(* CODESYS project PLC_Training_Estrusora_V3.project

Project tree, tasks and I/O mapping:
  Device : CODESYS Control Win V3 x64, CODESYS, version 3.5.21.40
    application Application
      libraries: Standard, 3.5.18.0 (System); VisuDialogs, * (System)
      task VISU_TASK (cyclic, interval 100 ms, priority 31) calls VisuElems.Visu_Prg
      task MainTask (cyclic, interval t#20ms, priority 1) calls PLC_Main
      function block FB_Inputs [LD]
      visualisation Visualization
      function block FB_Outputs [LD]
      function block FB_Process [LD]
      function block FB_Control [ST]
      function block FB_Events [ST]
      function block FB_PlantSim [ST]
      program PLC_Main [LD]
      global variables GVL_IO
      function block FB_Interlocks [LD]
      function block FB_Recipes [ST]
      text list TextList
      function block FB_LotHistory [ST]
      data type ST_LotRecord
  text list GlobalTextList
  text list System
  function block FB_Interlocks [LD]
*)

// Device/Application/ST_LotRecord
TYPE ST_LotRecord :
STRUCT
	LotNumber : DINT;
    RecipeID : INT;
    RecipeName : STRING[20];
    ProcessTime : TIME;
    MotorSpeed : INT;
    Completed : BOOL;
	CompletionDT : DT;
	TimestampText: STRING := DT_TO_STRING(CompletionDT);
END_STRUCT
END_TYPE

// Device/Application/GVL_IO
VAR_GLOBAL
	
    // =========================
    // RAW INPUTS (simulados / HMI)
    // =========================
	
    StartPB     : BOOL;   // Botón Start (RAW)
    StopPB_NC   : BOOL := TRUE;   // Botón Stop NC (RAW) -> TRUE = circuito OK, FALSE = presionado/abierto
	ResetPB     : BOOL;   // Boton de reset de falla
	LoadHopperPB : BOOL;  //Carga de la tolva
	AutoSelect : BOOL := TRUE;  // Boton del seleccion HMI
	ManualRunPB   : BOOL;  //Boton Arranque manual
	
    Sensor1     : BOOL;   // Sensor de Carga Minima (RAW)
	Sensor2		: BOOL;   //Sensor de carga media (RAW)
	Sensor3     : BOOL;   //Sensor de Carga Maxima (RAW)
	MotorFB     : BOOL;   // Feedback de motor/contactor (simulado)
	
	// =========================
    // NORMALIZED INPUTS (para lógica)
    // =========================
	
    Start       : BOOL;   // Evento/estado usable por lógica
    StopOK      : BOOL;   // TRUE = permitido (stop sano)
	ResetCmd       : BOOL;   // Reset de falla (simulado)
	ManualRunCmd  : BOOL; // Comando de arranque del motor
	LoadHopperCmd : BOOL; // Comando de carga de la tolva
	
	LevelLow    : BOOL;   // Sensor de carga de la tolva minima
	LevelMid    : BOOL;   // Sensor de carga de la tolva Media
	LevelHigh   : BOOL;   // Sensor de carga de la tolva Maximo
	
	// =========================
    // EVENTS (pulsos 1-scan)
    // =========================
	
    Start_Rise   : BOOL;   // Pulso flanco subida Start
    Stop_Fall   : BOOL;   // Pulso flanco bajada StopOK (o StopPB_NC si lo preferís)
	Reset_Rise  : BOOL;   // Pulso Subido para reset de falla.
	LoadHopper_Rise : BOOL; // Pulso Subida de carga de la tolva

	// =========================
    // MODOS / CONTROL
    // =========================
	
	AutoMode : BOOL := TRUE;
	ManualMode : BOOL := FALSE;

	RunCmd       : BOOL;     // Comando general de marcha
	State : INT := 0;        // 0= IDLE, 5=Manual, 10=STARTING, 20=Processing, 40=Complete 90=FAULT
	StateText : STRING[50];	 // almacena la cadena segun estado
	StateProcessing : BOOL;  //Badera de control de estado
	BatchComplete : BOOL;    //Indicador del final del proceso
	
	//==========================
	//Codigos de falla Y alarmas
	//=========================
	
	Fault        : BOOL;  // Falla activa (latch)
	FaultCode_MotorNoStart : BOOL; 
	FaultCode_LevelInvalid : BOOL; 
	
	Alarm_NoMaterial_Latched : BOOL; // Latch de control de Alarmas
	Alarm_NoMaterialStart : BOOL;
	AlarmText : STRING[50];
	
    // =========================
    // OUTPUTS (lógicos)
    // =========================
	
	AlarmLamp    : BOOL;  // Lámpara/alarma (lógico Rojo)
    MotorCmd     : BOOL;  // Comando a motor (lógico)
    ReadyLamp    : BOOL;   // Lampara de Maquina Lista para correr (Logico Amarillo)
	
	//==========================
	// Simulacion / Proceso
	//==========================
	
	SimEnable  : BOOL := TRUE;   // habilita simulación de planta
    MotorAngle : INT  := 0;      // 0..359 (para animación)
	ProcessTimeA : TIME ;  //Tiempo del proceso por receta.
	CantLotesProc   : DINT;      //Cuenta la cantidad de lotes procesados
	VelocidadMotor : INT; //Velocidad de giro del motor
	
	//==========================
	//Interlocks
	//==========================
	
	StartPermissive : BOOL ;
	RunPermissive : BOOL ;
	LoadPermissive : BOOL;
	ResetPermissive : BOOL;
	Ready       : BOOL;   // Comando de inicio.
	RecipeChangePermissive: BOOL ; // Limita el cambio de receta durante una corrida.
	
	//==========================
	//Recetas (Variables)
	//==========================

	RecipeSelected : INT; //Recibe la opcion seleccionada
	RecipeID : INT ; //Identificador de la receta.
	RecipeName : STRING[20]; // Recibe el nombre de la receta
	
	//==========================
	//Historial de lotes y fallas
	//==========================
	
	LotHistory : ARRAY[1..20] OF ST_lotRecord;
	LotHistoryIndex : INT := 1;	
	TimestampText : STRING[30];
	LastLotTimestampText : STRING[30];
	LotHistoryCount : INT ;
	
END_VAR

// Device/Application/PLC_Main
PROGRAM PLC_Main
VAR
	fbInputs: FB_Inputs;
	fbEvents: FB_Events;
	fbControl: FB_Control;
	fbProcess: FB_Process;
	fbOutputs: FB_Outputs;
	fbPlantSim: FB_PlantSim;
	fbInterlocks: FB_Interlocks;
	fbRecipes: FB_Recipes;
	fbLotHistory: FB_LotHistory;
	
	VarTimeCur : DT;
	
	Reloj: RTC;
END_VAR

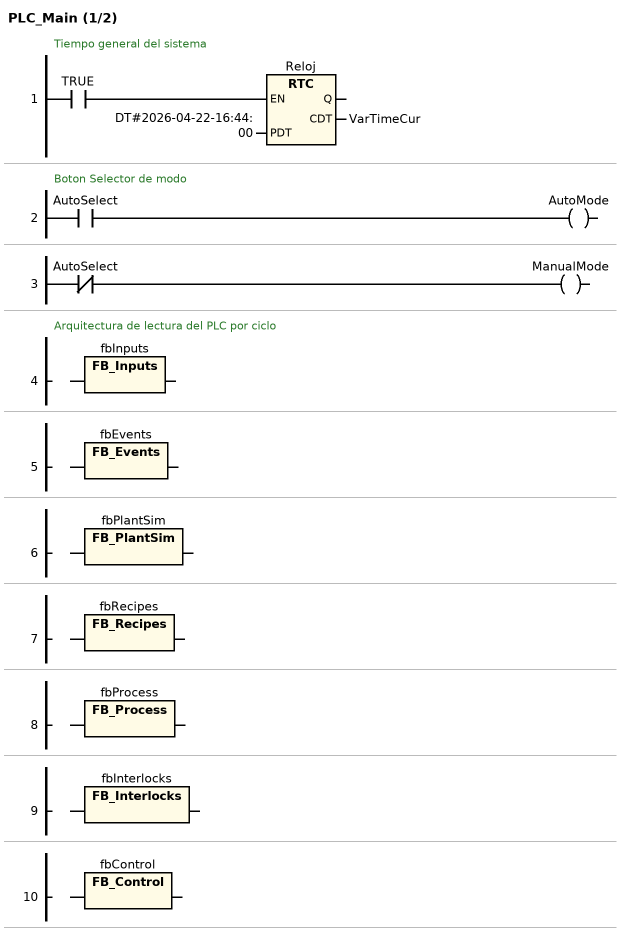
// NETWORK 1
// Tiempo general del sistema
Reloj(EN := TRUE, PDT := DT#2026-04-22-16:44:00, CDT => VarTimeCur); // RTC

// NETWORK 2
// Boton Selector de modo
AutoMode := AutoSelect;

// NETWORK 3
ManualMode := NOT AutoSelect;

// NETWORK 4
// Arquitectura de lectura del PLC por ciclo
fbInputs(); // FB_Inputs

// NETWORK 5
fbEvents(); // FB_Events

// NETWORK 6
fbPlantSim(); // FB_PlantSim

// NETWORK 7
fbRecipes(); // FB_Recipes

// NETWORK 8
fbProcess(); // FB_Process

// NETWORK 9
fbInterlocks(); // FB_Interlocks

// NETWORK 10
fbControl(); // FB_Control

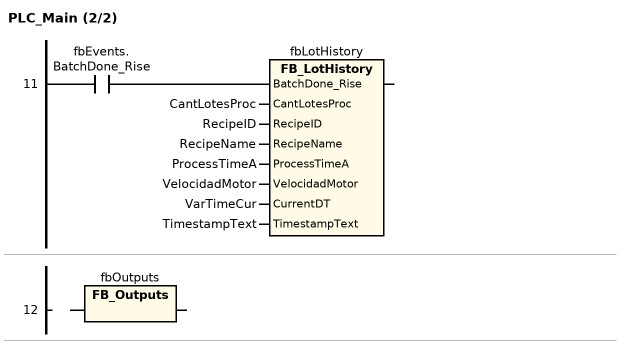
// NETWORK 11
fbLotHistory(
    BatchDone_Rise := fbEvents.BatchDone_Rise,
    CantLotesProc := CantLotesProc,
    RecipeID := RecipeID,
    RecipeName := RecipeName,
    ProcessTimeA := ProcessTimeA,
    VelocidadMotor := VelocidadMotor,
    CurrentDT := VarTimeCur,
    TimestampText := TimestampText); // FB_LotHistory

// NETWORK 12
fbOutputs(); // FB_Outputs

END_PROGRAM

// Device/Application/FB_Inputs
FUNCTION_BLOCK FB_Inputs
VAR_INPUT
END_VAR
VAR_OUTPUT
END_VAR
VAR
END_VAR

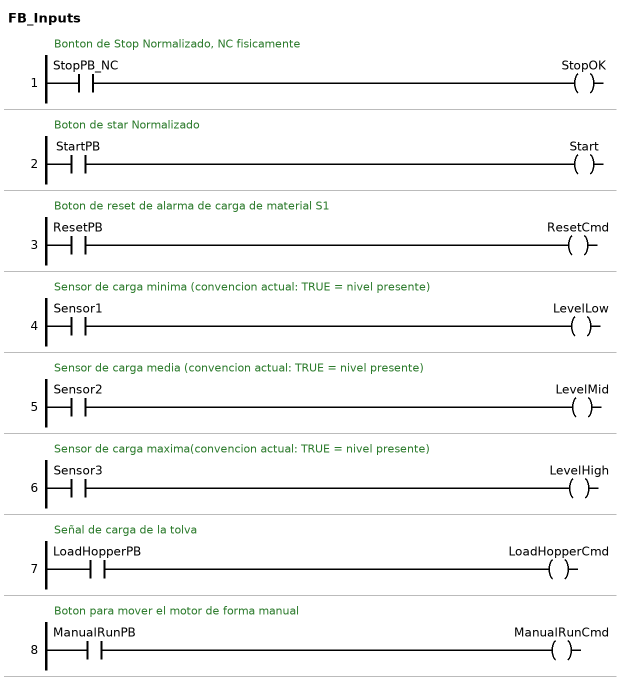
// NETWORK 1
// Bonton de Stop Normalizado, NC fisicamente
StopOK := StopPB_NC;

// NETWORK 2
// Boton de star Normalizado
Start := StartPB;

// NETWORK 3
// Boton de reset de alarma de carga de material S1
ResetCmd := ResetPB;

// NETWORK 4
// Sensor de carga minima (convencion actual: TRUE = nivel presente)
LevelLow := Sensor1;

// NETWORK 5
// Sensor de carga media (convencion actual: TRUE = nivel presente)
LevelMid := Sensor2;

// NETWORK 6
// Sensor de carga maxima(convencion actual: TRUE = nivel presente)
LevelHigh := Sensor3;

// NETWORK 7
// Señal de carga de la tolva
LoadHopperCmd := LoadHopperPB;

// NETWORK 8
// Boton para mover el motor de forma manual
ManualRunCmd := ManualRunPB;

END_FUNCTION_BLOCK

// Device/Application/FB_Events
FUNCTION_BLOCK FB_Events
VAR_INPUT
END_VAR
VAR_OUTPUT
	BatchDone_Rise : BOOL;
END_VAR
VAR
	
	rStart: R_TRIG;
	fStop: F_TRIG;
	rReset: R_TRIG;
	rBatchDone: R_TRIG;
	rloadHopper: R_TRIG;
	rsNoMaterial : RS;
	rsNoStop : RS;

END_VAR

// Flanco de subida en Start
rStart(CLK := Start);
Start_Rise := rStart.Q;

// Flanco de bajada en StopOK
fStop(CLK := StopOK);
Stop_Fall := fStop.Q;

//Flaco de subida Reset Fault
rReset(CLK := resetCmd);
Reset_Rise := rReset.Q;

//Flaco de subida estado 40 a 20 (Conteo de lotes)
rBatchDone(CLK := BatchComplete);
BatchDone_Rise := rBatchDone.Q;

IF BatchDone_Rise THEN
	CantlotesProc := CantlotesProc + 1;
	
END_IF;

//Flaco de Carga de la Tolva

rLoadHopper(CLK := LoadHopperCmd);
LoadHopper_Rise := rLoadHopper.Q;

// Alarma de arranque sin material
Alarm_NoMaterialStart := Start_Rise AND StopOK AND NOT LevelMid;

// Latch de alarma
rsNoMaterial(
    SET := Alarm_NoMaterialStart,
    RESET1 := Reset_Rise OR LevelMid
);

Alarm_NoMaterial_Latched := rsNoMaterial.Q1;

// Mensaje HMI

IF Alarm_NoMaterial_Latched THEN
    AlarmText := 'START BLOQUEADO: CARGAR MATERIAL';
ELSIF NOT StopOK THEN
    AlarmText := 'START BLOQUEADO: ACTIVAR STOP';
ELSE
    AlarmText := '';
END_IF;

END_FUNCTION_BLOCK

// Device/Application/FB_PlantSim
FUNCTION_BLOCK FB_PlantSim
VAR_INPUT
END_VAR
VAR_OUTPUT
END_VAR
VAR
	tContactor : TON;   // retardo para feedback de motor
	
	//Simulacion Nivel de material
	tConsumeHigh : TON;
	tConsumeMid : TON;
	tConsumeLow : TON;
	
	
END_VAR

// Si no hay simulación, no tocamos nada
IF NOT SimEnable THEN
    MotorFB := FALSE;
    RETURN;
END_IF;

// -------------------------
// Simulación de MotorFB (contactor)
// MotorCmd -> después de 300ms MotorFB = TRUE
// -------------------------
tContactor(IN := MotorCmd, PT := T#300MS);
IF MotorCmd THEN
    MotorFB := tContactor.Q;
ELSE
    MotorFB := FALSE;
END_IF;

// -------------------------
// "Animación" simple: ángulo del motor
// (solo para visualizar movimiento)
// -------------------------
IF MotorFB THEN
    MotorAngle := MotorAngle + VelocidadMotor;   // velocidad visual
    IF MotorAngle >= 360 THEN
        MotorAngle := MotorAngle - 360;
    END_IF;
END_IF;

//--------------------------
//Carga de la tova
//--------------------------

IF LoadHopper_Rise AND LoadPermissive THEN
	
	Sensor1 := TRUE;
	Sensor2 := TRUE;
	Sensor3 := TRUE;
	
END_IF;

//--------------------------
//Sumulacion de consumo de material en tolva
//Solo Descarga durante PROSSESING con motor confirmado.
//---------------------------

tConsumeHigh(IN := StateProcessing AND MotorFB, PT := T#2S);
tConsumeMid(IN := StateProcessing AND MotorFB, PT := T#4S);
tConsumeLow(IN := StateProcessing AND MotorFB, PT := T#6S);

//Proceso de consumo segun TON
IF StateProcessing AND MotorFB THEN

	IF tConsumeHigh.Q THEN
		Sensor3 := FALSE;
	END_IF;
	
	IF tConsumeMid.Q THEN
		Sensor2 := FALSE;
	END_IF;
	
	IF tConsumeLow.Q THEN
		Sensor1 := FALSE;
	END_IF;

END_IF;

END_FUNCTION_BLOCK

// Device/Application/FB_Recipes
FUNCTION_BLOCK FB_Recipes
VAR_INPUT
END_VAR
VAR_OUTPUT
END_VAR
VAR
	RecipeLatched : INT := 1;
END_VAR

//Seleccionador de Recetas del proceso

IF RecipeChangePermissive THEN
    RecipeLatched := RecipeSelected;
END_IF;

CASE RecipeLatched OF
	
	1:
		RecipeID := 1;
		RecipeName := 'Normal';
		ProcessTimeA := T#5S;
		VelocidadMotor := 3;
	2:
		RecipeID := 2;
		RecipeName := 'Rapida';
		ProcessTimeA := T#4S;
		VelocidadMotor := 4;
	ELSE
		RecipeID := 0;
		RecipeName := 'Simulacion';
		ProcessTimeA := T#6S;
		VelocidadMotor := 2;
	
END_CASE;

END_FUNCTION_BLOCK

// Device/Application/FB_Process
FUNCTION_BLOCK FB_Process
VAR_INPUT
END_VAR
VAR_OUTPUT
END_VAR
VAR
	
	//Temporizadores
	tNoSensor : TON;
	Monitor: TIME;
	tMotorStart : TON;
	Mrespuesta: TIME;
	tBatchProcess: TON;
	BatchMonitor: TIME;
	
	//Memorias Biestables
	rsNoSensor: RS;
	rsMotorNoMotor: Rs;
	rsLevelInvalid: RS;
	
END_VAR

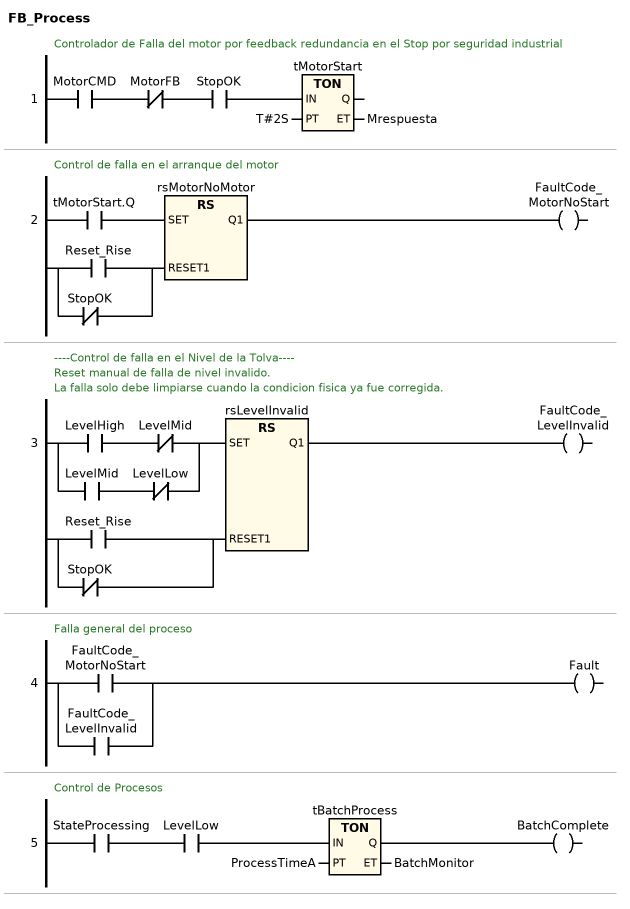
// NETWORK 1
// Controlador de Falla del motor por feedback redundancia en el Stop por seguridad industrial
tMotorStart(IN := MotorCMD AND NOT MotorFB AND StopOK, PT := T#2S, ET => Mrespuesta); // TON

// NETWORK 2
// Control de falla en el arranque del motor
rsMotorNoMotor(SET := tMotorStart.Q, RESET1 := Reset_Rise OR NOT StopOK); // RS
FaultCode_MotorNoStart := rsMotorNoMotor.Q1;

// NETWORK 3
// ----Control de falla en el Nivel de la Tolva----
//
// Reset manual de falla de nivel invalido.
// La falla solo debe limpiarse cuando la condicion fisica ya fue corregida.
rsLevelInvalid(SET := LevelHigh AND NOT LevelMid OR LevelMid AND NOT LevelLow, RESET1 := Reset_Rise OR NOT StopOK); // RS
FaultCode_LevelInvalid := rsLevelInvalid.Q1;

// NETWORK 4
// Falla general del proceso
Fault := FaultCode_MotorNoStart OR FaultCode_LevelInvalid;

// NETWORK 5
// Control de Procesos
tBatchProcess(IN := StateProcessing AND LevelLow, PT := ProcessTimeA, ET => BatchMonitor); // TON
BatchComplete := tBatchProcess.Q;

END_FUNCTION_BLOCK

// Device/Application/FB_Interlocks
FUNCTION_BLOCK FB_Interlocks
VAR_INPUT
END_VAR
VAR_OUTPUT
END_VAR
VAR
	StateIdle : BOOL;
	StateComplete : BOOL;
END_VAR

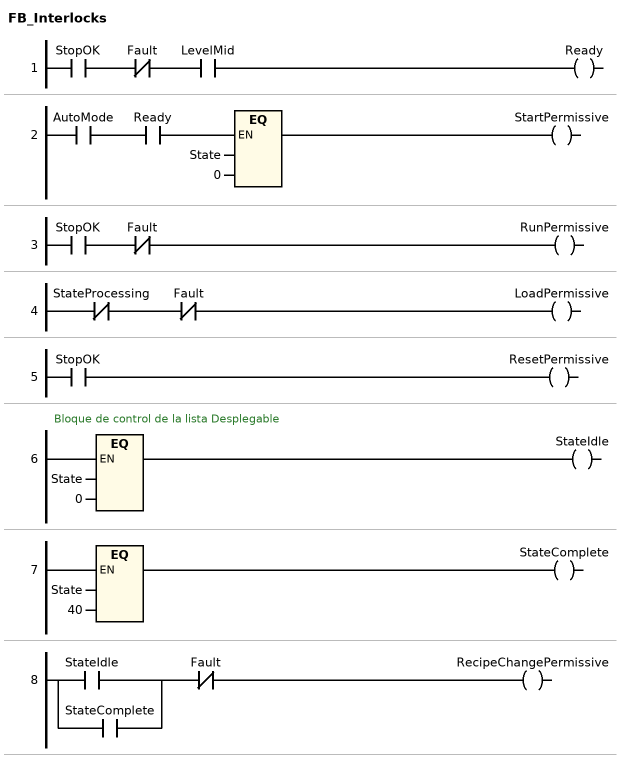
// NETWORK 1
Ready := StopOK AND NOT Fault AND LevelMid;

// NETWORK 2
StartPermissive := AutoMode AND Ready AND State = 0;

// NETWORK 3
RunPermissive := StopOK AND NOT Fault;

// NETWORK 4
LoadPermissive := NOT StateProcessing AND NOT Fault;

// NETWORK 5
ResetPermissive := StopOK;

// NETWORK 6
// Bloque de control de la lista Desplegable
StateIdle := State = 0;

// NETWORK 7
StateComplete := State = 40;

// NETWORK 8
RecipeChangePermissive := (StateIdle OR StateComplete) AND NOT Fault;

END_FUNCTION_BLOCK

// FB_Interlocks
FUNCTION_BLOCK FB_Interlocks
VAR_INPUT
END_VAR
VAR_OUTPUT
END_VAR
VAR
END_VAR

// NETWORK 1

END_FUNCTION_BLOCK

// Device/Application/FB_Control
FUNCTION_BLOCK FB_Control
VAR_INPUT
END_VAR
VAR_OUTPUT
END_VAR
VAR
END_VAR

// ---------------------------------------------------------
// Maquina de estados principal
// 0  = IDLE
// 5  = MANUAL
// 10 = STARTING
// 20 = RUNNING
// 40 = PROCESSING
// 90 = FAULT
// ---------------------------------------------------------

// Valor por defecto
RunCmd := FALSE;
StateProcessing := FALSE;

// Seleccion de modo

IF ManualMode THEN
    // Modo Manual
	
    IF Fault THEN
        State := 90;
        StateText := 'FAULT';

    ELSE
        State := 5;
        StateText := 'En Manual';

        IF RunPermissive AND ManualRunCmd THEN
            RunCmd := TRUE;
        END_IF;

    END_IF;

ELSE
	
//Modo Automatico	

	// Falla global con prioridad
    IF Fault AND (State <> 90) THEN
        State := 90;
    END_IF;
	
    CASE State OF

        0: // IDLE
            StateText := 'IDLE';

            IF StartPermissive AND Start_Rise THEN
                State := 10;
            END_IF;

        10: // STARTING
            RunCmd := TRUE;
            StateText := 'STARTING';

            IF NOT StopOK THEN
                State := 0;

            ELSIF MotorFB THEN
                State := 20;
            END_IF;

        20: // PROCESSING
            RunCmd := TRUE;
			StateProcessing := TRUE;
			StateText := 'PROCESSING';

            IF NOT StopOK THEN
                State := 0;
				
			ELSIF NOT LevelLow THEN
				State := 90;
				
			ELSIF BatchComplete THEN
				State := 40;
				
            END_IF;
			
		40: // COMPLETE
			StateText := 'COMPLETE';
			
			IF Reset_Rise THEN
				State := 0;
			END_IF;	

        90: // FAULT
            StateText := 'FAULT';

            IF FaultCode_MotorNoStart AND NOT FaultCode_LevelInvalid THEN
                StateText := 'Motor Fault';

            ELSIF FaultCode_LevelInvalid AND NOT FaultCode_MotorNoStart THEN
                StateText := 'Level Fault';

            ELSIF FaultCode_LevelInvalid AND FaultCode_MotorNoStart THEN
                StateText := 'Multi FAULT';	
            END_IF;

            IF ResetPermissive AND Reset_Rise AND NOT Fault THEN
                State := 0;
            END_IF;
            
			

    ELSE
        State := 0;
        StateText := 'UNKNOWN';

    END_CASE;

END_IF;

END_FUNCTION_BLOCK

// Device/Application/FB_LotHistory
FUNCTION_BLOCK FB_LotHistory
VAR_INPUT
	BatchDone_Rise : BOOL;
    CantLotesProc : DINT;
    RecipeID : INT;
    RecipeName : STRING[20];
    ProcessTimeA : TIME;
    VelocidadMotor : INT;
	CurrentDT : DT;
	TimestampText: STRING[30];
END_VAR
VAR_OUTPUT
END_VAR
VAR
END_VAR

//Memoria temporal de procesos y lotes

//Manejo de indice circular maximo 20 espacios de guardado
IF BatchDone_Rise THEN

IF LotHistoryCount < 20 THEN
    LotHistoryCount := LotHistoryCount + 1;
END_IF;
	
IF LotHistoryIndex < 20 THEN
	
	LotHistoryIndex := LotHistoryIndex + 1;
	
ELSE
	
	LotHistoryIndex := 1;
	
	
END_IF;
	
	LotHistory[LotHistoryIndex].LotNumber := CantLotesProc;
	LotHistory[LotHistoryIndex].RecipeID := RecipeID;
    LotHistory[LotHistoryIndex].RecipeName := RecipeName;
    LotHistory[LotHistoryIndex].ProcessTime := ProcessTimeA;
    LotHistory[LotHistoryIndex].MotorSpeed := VelocidadMotor;
    LotHistory[LotHistoryIndex].Completed := TRUE;
	LotHistory[LotHistoryIndex].CompletionDT := CurrentDT;
	LotHistory[LotHistoryIndex].TimestampText := DT_TO_STRING(CurrentDT);
	LastLotTimestampText := LotHistory[LotHistoryIndex].TimestampText;


	
END_IF;

END_FUNCTION_BLOCK

// Device/Application/FB_Outputs
FUNCTION_BLOCK FB_Outputs
VAR_INPUT
END_VAR
VAR_OUTPUT
END_VAR
VAR
END_VAR

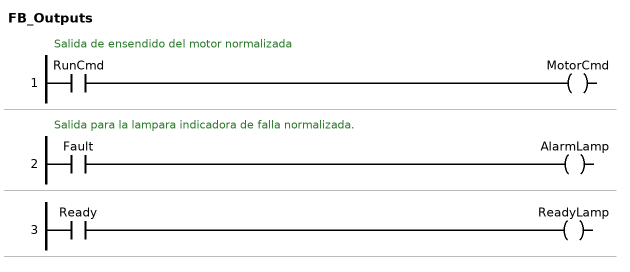
// NETWORK 1
// Salida de ensendido del motor normalizada
MotorCmd := RunCmd;

// NETWORK 2
// Salida para la lampara indicadora de falla normalizada.
AlarmLamp := Fault;

// NETWORK 3
ReadyLamp := Ready;

END_FUNCTION_BLOCK

// Device/Application/Visualization
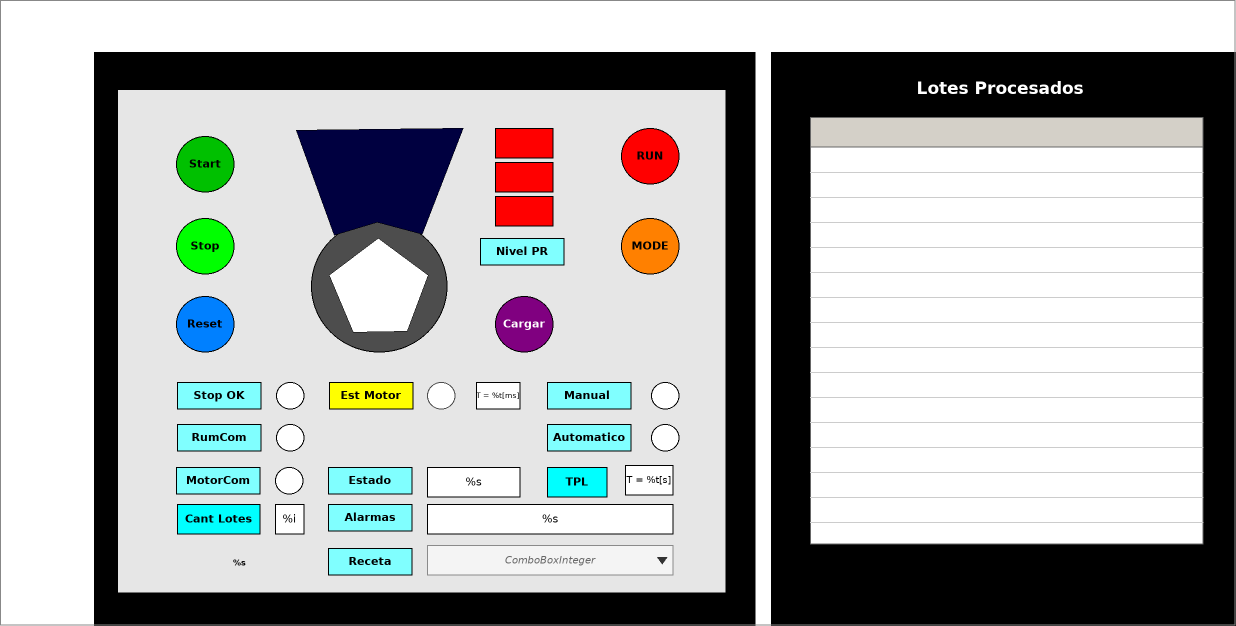
VISUALIZATION Visualization  // 1236x626
    Rectangle (771,52 465x574)
    Rectangle (94,52 661x574)
    Rectangle (117,89 609x504)
        tap ManualMode
    Ellipse (311,220 136x132), colour toggle: FaultCode_MotorNoStart
    Ellipse (176,136 58x56), "Start", colour toggle: Start
        tap StartPB
    Ellipse (176,218 58x56), "Stop", colour toggle: StopPB_NC
        tap StopPB_NC p1329445385=TRUE
    Ellipse (176,296 58x56), "Reset", colour toggle: ResetPB
        tap ResetPB
    Rectangle (177,382 84x27), "Stop OK"
    Ellipse (276,382 28x27), colour toggle: StopOK
    Rectangle (177,424 84x27), "RumCom"
    Ellipse (276,424 28x27), colour toggle: RunCmd
    Rectangle (176,467 84x27), "MotorCom"
    Ellipse (275,467 28x27), colour toggle: MotorCmd
    Rectangle (329,382 84x27), "Est Motor"
    Ellipse (427,382 28x27), colour toggle: SimEnable
        toggle SimEnable
    Rectangle (328,467 84x27), "Estado"
    Rectangle (476,382 44x27), "T = %t[ms]", text variable: PLC_Main.fbProcess.Mrespuesta
    Polygon (329,275) (378,238) (428,275) (407,331) (353,332)
        p2858320360: MotorAngle
    Polygon (334,235) (296,130) (463,128) (422,234) (377,222), colour toggle: FaultCode_LevelInvalid
    Label (581,119 92x30)
    RoundedRectangle (427,467 93x30), "%s", text variable: StateText
    Rectangle (547,382 84x27), "Manual"
    Rectangle (547,424 84x27), "Automatico"
    Ellipse (651,382 28x27), colour toggle: ManualMode
    Ellipse (651,424 28x27), colour toggle: AutoMode
    Ellipse (621,128 58x56), "RUN", colour toggle: RunCmd
        tap ManualRunPB
    Ellipse (621,218 58x56), "MODE", colour toggle: AutoSelect
        toggle AutoSelect
    Rectangle (177,504 83x30), "Cant Lotes"
    Rectangle (275,504 29x30), "%i", text variable: CantLotesProc
    Rectangle (625,465 48x30), "T = %t[s]", text variable: PLC_Main.fbProcess.BatchMonitor
    Rectangle (547,467 60x30), "TPL"
    Rectangle (495,128 58x30), colour toggle: LevelHigh
    Rectangle (495,162 58x30), colour toggle: LevelMid
    Rectangle (495,196 58x30), colour toggle: LevelLow
    Rectangle (480,238 84x27), "Nivel PR"
    Ellipse (495,296 58x56), "Cargar", colour toggle: LoadHopperCmd
        tap LoadHopperPB
    Rectangle (328,504 84x27), "Alarmas"
    RoundedRectangle (427,504 246x30), "%s", text variable: AlarmText
    ComboBoxInteger (427,545 246x30), variable: RecipeSelected, text list: 'TextList'
    Rectangle (328,548 84x27), "Receta"
    RoundedRectangle (176,548 127x30), "%s", text variable: LastLotTimestampText
    Table (810,117 393x427), data array: LotHistory
        p3854506369: LotHistory[INDEX].LotNumber
        p1892666644: LotHistory[INDEX].RecipeID
        p338671338: LotHistory[INDEX].RecipeName
        p2170511999: LotHistory[INDEX].ProcessTime
        p3723444502: LotHistory[INDEX].MotorSpeed
        p1218418051: LotHistory[INDEX].Completed
        p746581629: LotHistory[INDEX].CompletionDT
        p3104783080: LotHistory[INDEX].TimestampText
        p2232123230: Lote
        p1755163831: Receta
        p4092479075: Tiempo
        p2237128397: Velocidad
        p4088588272: Fecha
        p1014161805: 20 - 1 + INT#1
        p1128707560: LotHistoryCount +1
    RoundedRectangle (895,73 210x30), "Lotes Procesados"
END_VISUALIZATION

(* text list System (id | default)
  Apr | Apr
  April | April
  Aug | Aug
  August | August
  Dec | Dec
  December | December
  Feb | Feb
  February | February
  Fri | Fri
  Friday | Friday
  Jan | Jan
  January | January
  Jul | Jul
  July | July
  Jun | Jun
  June | June
  Mar | Mar
  March | March
  May | May
  May_3Letter | May
  Mon | Mon
  Monday | Monday
  Nov | Nov
  November | November
  Oct | Oct
  October | October
  Sat | Sat
  Saturday | Saturday
  Sep | Sep
  September | September
  Sun | Sun
  Sunday | Sunday
  Thu | Thu
  Thursday | Thursday
  Tue | Tue
  Tuesday | Tuesday
  Wed | Wed
  Wednesday | Wednesday
   |  *)

(* text list TextList (id | default)
  1 | Duracion Normal
  2 | Receta Rapida
  0 | Simulacion
   |  *)
